// Mitsubishi GX Works2 project: 42015010_0528 (1)   PLC: Q02/Q02H

PROGRAM MAIN
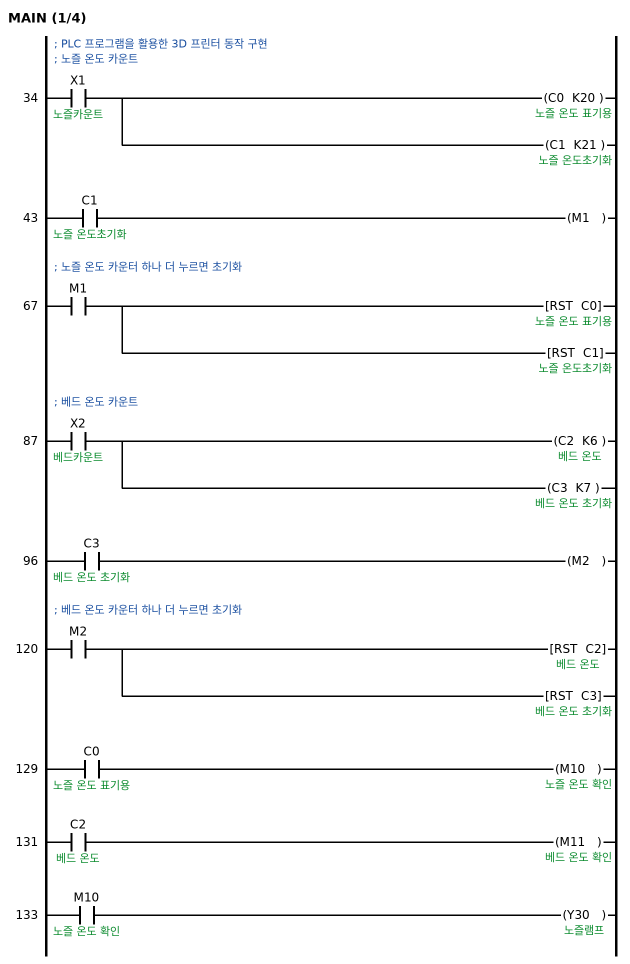
; PLC 프로그램을 활용한 3D 프린터 동작 구현
; 노즐 온도 카운트
34    LD      X1  ; 노즐카운트
      OUT     C0 K20  ; 노즐 온도 표기용
      OUT     C1 K21  ; 노즐 온도초기화
43    LD      C1  ; 노즐 온도초기화
      OUT     M1
; 노즐 온도 카운터 하나 더 누르면 초기화
67    LD      M1
      RST     C0  ; 노즐 온도 표기용
      RST     C1  ; 노즐 온도초기화
; 베드 온도 카운트
87    LD      X2  ; 베드카운트
      OUT     C2 K6  ; 베드 온도
      OUT     C3 K7  ; 베드 온도 초기화
96    LD      C3  ; 베드 온도 초기화
      OUT     M2
; 베드 온도 카운터 하나 더 누르면 초기화
120   LD      M2
      RST     C2  ; 베드 온도
      RST     C3  ; 베드 온도 초기화
129   LD      C0  ; 노즐 온도 표기용
      OUT     M10  ; 노즐 온도 확인
131   LD      C2  ; 베드 온도
      OUT     M11  ; 베드 온도 확인
133   LD      M10  ; 노즐 온도 확인
      OUT     Y30  ; 노즐램프
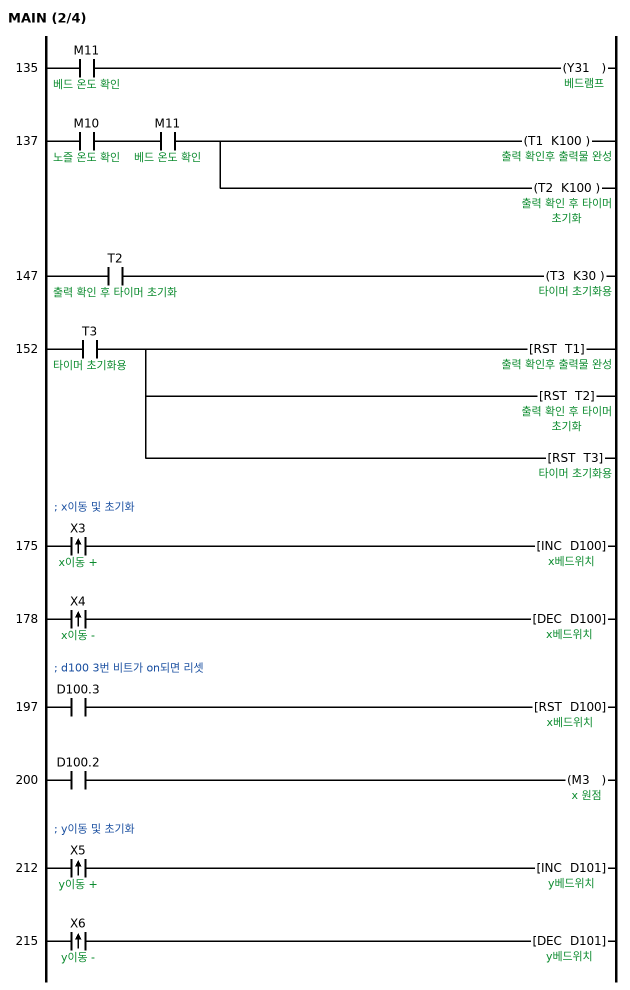
135   LD      M11  ; 베드 온도 확인
      OUT     Y31  ; 베드램프
137   LD      M10  ; 노즐 온도 확인
      AND     M11  ; 베드 온도 확인
      OUT     T1 K100  ; 출력 확인후 출력물 완성
      OUT     T2 K100  ; 출력 확인 후 타이머 초기화
147   LD      T2  ; 출력 확인 후 타이머 초기화
      OUT     T3 K30  ; 타이머 초기화용
152   LD      T3  ; 타이머 초기화용
      RST     T1  ; 출력 확인후 출력물 완성
      RST     T2  ; 출력 확인 후 타이머 초기화
      RST     T3  ; 타이머 초기화용
; x이동 및 초기화
175   LDP     X3  ; x이동 +
      INC     D100  ; x베드위치
178   LDP     X4  ; x이동 -
      DEC     D100
; d100 3번 비트가 on되면 리셋
197   LD      D100.3
      RST     D100  ; x베드위치
200   LD      D100.2
      OUT     M3  ; x 원점
; y이동 및 초기화
212   LDP     X5  ; y이동 +
      INC     D101  ; y베드위치
215   LDP     X6  ; y이동 -
      DEC     D101
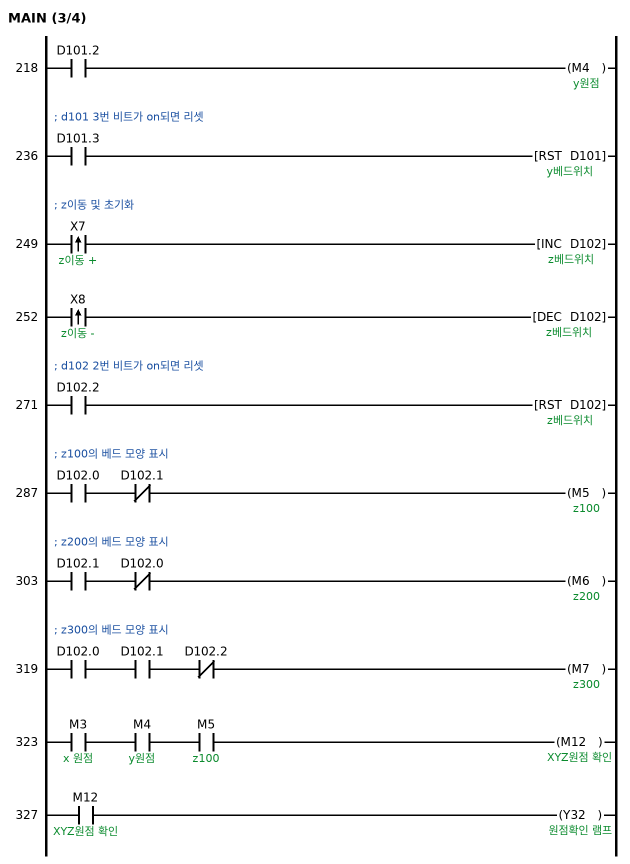
218   LD      D101.2
      OUT     M4  ; y원점
; d101 3번 비트가 on되면 리셋
236   LD      D101.3
      RST     D101  ; y베드위치
; z이동 및 초기화
249   LDP     X7  ; z이동 +
      INC     D102  ; z베드위치
252   LDP     X8  ; z이동 -
      DEC     D102
; d102 2번 비트가 on되면 리셋
271   LD      D102.2
      RST     D102  ; z베드위치
; z100의 베드 모양 표시
287   LD      D102.0
      ANI     D102.1
      OUT     M5  ; z100
; z200의 베드 모양 표시
303   LD      D102.1
      ANI     D102.0
      OUT     M6  ; z200
; z300의 베드 모양 표시
319   LD      D102.0
      AND     D102.1
      ANI     D102.2
      OUT     M7  ; z300
323   LD      M3  ; x 원점
      AND     M4  ; y원점
      AND     M5  ; z100
      OUT     M12  ; XYZ원점 확인
327   LD      M12  ; XYZ원점 확인
      OUT     Y32  ; 원점확인 램프
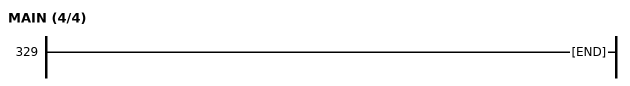
329   END
END_PROGRAM
